(* IEC 61131-3 sources: ErrorLib/src/Ar/Diagnostics/ErrorProg, 3 files *)

(* ---- ErrorProg.typ ---- *)
(*
* File: ErrorProg.typ
* Copyright (c) 2023 Loupe
* https://loupe.team
*
* This file is part of ErrorProg, licensed under the MIT License.
*)

TYPE

END_TYPE

(* ---- ErrorProgCyclic.st ---- *)
(*
* File: ErrorProgCyclic.st
* Copyright (c) 2023 Loupe
* https://loupe.team
*
* This file is part of ErrorProg, licensed under the MIT License.
*)

PROGRAM _CYCLIC

ErrorCollectorFn_HMI_Cyclic( gErrorCollectorHMI, gErrorCollector );

ErrorCollectorFn_Cyclic( gErrorCollector );

END_PROGRAM

(* ---- ErrorProgInit.st ---- *)
(*
* File: ErrorProgInit.st
* Copyright (c) 2023 Loupe
* https://loupe.team
*
* This file is part of ErrorProg, licensed under the MIT License.
*)

PROGRAM _INIT

(* gErrorCollector is initialized in FirstInitProg - Init only if it hasn't already been *)
	IF NOT gErrorCollector.Internal.Initialized THEN
		ErrorCollectorFn_Init(gErrorCollector);
	END_IF
(* Sources are added to gErrorCollector in the source program. *)

END_PROGRAM
